// SIMATIC S7-200 project (STEP 7-Micro/WIN), CPU 224XP REL 02.01

ORGANIZATION_BLOCK MAIN:OB1
TITLE=PROGRAM COMMENTS
BEGIN
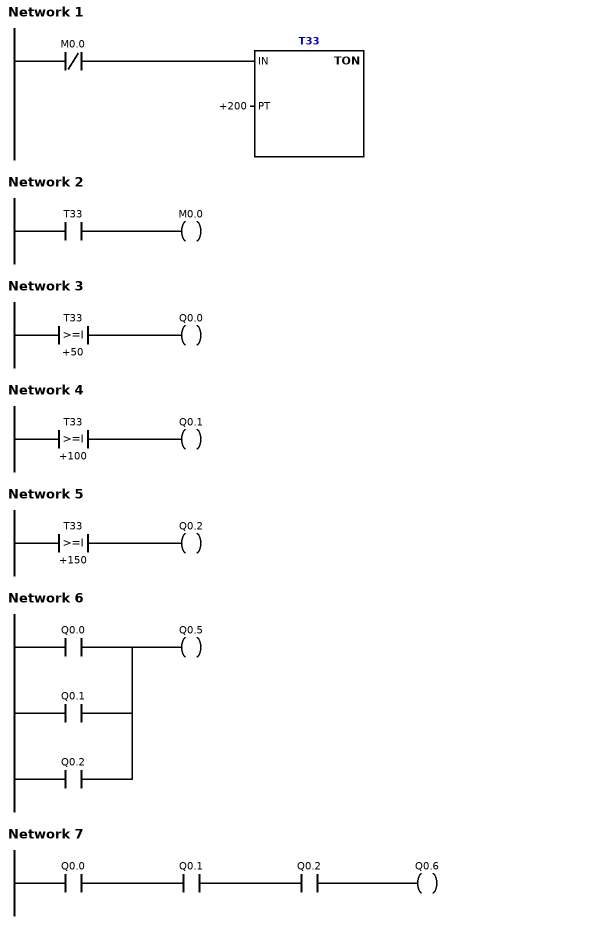
Network 1
// (network saved uncompiled; LAD cells follow)
// row 0: c0 -|/|- M0.0  c1 --  c2 [TON T33 IN:=power@row0, PT:=+200]
// row 1: c2 [box]
Network 2
LD     T33
=      M0.0
Network 3
LDW>=  T33, +50
=      Q0.0
Network 4
LDW>=  T33, +100
=      Q0.1
Network 5
LDW>=  T33, +150
=      Q0.2
Network 6
LD     Q0.0
O      Q0.1
O      Q0.2
=      Q0.5
Network 7
LD     Q0.0
A      Q0.1
A      Q0.2
=      Q0.6
END_ORGANIZATION_BLOCK
